(* Logix 5000 project; controller Bandas_Divert_Merge Emulate 5570 rev 30.12; software revision 30.00 *)

TASK MainTask (continuous, watchdog 500 ms) : MainProgram

MODULES
   Local : Emulate 5570 (ICP 2, rev 30.12)
      VIRTUAL_OUTPUTS : vendor 1 type 0 code 15 (ICP 4, rev 1.1, Output RPI 50 ms)   // Salidas_PLC_Bandas
      VIRTUAL_INPUTS : vendor 1 type 0 code 15 (ICP 3, rev 1.1, Output RPI 50 ms)   // Entradas_PLC_Bandas_Transportadoras
END_MODULES

VAR_GLOBAL   (* controller tags *)
   B1 : BOOL;
   B11 : BOOL;
   B2A : BOOL;
   B2A1 : BOOL;   // Banda hacia arriba
   B2B : BOOL;
   B2B1 : BOOL;   // Banda hacia izquierda
   B4A : BOOL;   // Banda4A
   B4B : BOOL;   // Banda4B
   B6A : BOOL;   // banda6A
   B6B : BOOL;   // banda 6b
   B_decA : BOOL;
   B_decB : BOOL;
   B_secA : BOOL;
   B_secB : BOOL;
   P : BOOL;   // Selector de baldosas
   Press_ActLX : INT;
   Press_ActLY : INT;
   Press_CilinderMax : BOOL;
   Press_CilinderMin : BOOL;
   Press_CilinderPos : INT;
   Press_FillerMax : BOOL;
   Press_FillerMin : BOOL;
   Press_FillerPos : INT;
   Press_Manguera : BOOL;
   Press_SourceTiles : BOOL;
   Press_SXmax : BOOL;
   Press_SXmin : BOOL;
   Press_TileMax : BOOL;
   Press_TileMin : BOOL;
   Press_TilePos : INT;
   Press_Ymax : BOOL;
   Press_Ymin : BOOL;
   S1 : BOOL;
   S11 : BOOL;
   S2 : BOOL;
   S21 : BOOL;
   S4 : BOOL;   // Sensor4_Para la engobadora
   S6 : BOOL;   // Sensor6_Va para el merge
   S_dec : BOOL;
   S_sec : BOOL;
   SFC_Bder4 : BOOL;
   SFC_Bizq4 : BOOL;
   SFC_BunionX : BOOL;
   SFC_BunionY : BOOL;
   SFC_Sder4 : BOOL;
   SFC_Sizq4 : BOOL;
   SFC_Sunion : BOOL;
   Start : BOOL;
   Tipper_Grab : INT;
   Tipper_Rollers : BOOL;
   Tipper_Rotate : INT;
   Tipper_S1 : BOOL;
   Tipper_S2 : BOOL;
END_VAR

PROGRAM MainProgram   (* main routine MainRoutine *)
VAR
   Action_000 : SFC_ACTION := (Status := 16#0020_0000, PauseTimer := 1);
   Action_001 : SFC_ACTION := (Status := 16#0020_0000, PauseTimer := 1);
   Action_002 : SFC_ACTION := (Status := 16#0020_0000, PauseTimer := 1);
   Action_003 : SFC_ACTION := (Status := 16#0020_0000, PauseTimer := 1);
   Action_004 : SFC_ACTION := (Status := 16#0020_0000, PauseTimer := 1);
   Action_005 : SFC_ACTION := (Status := 16#0020_0000, PauseTimer := 1);
   Action_006 : SFC_ACTION := (Status := 16#0020_0000, PauseTimer := 1);
   Action_007 : SFC_ACTION := (Status := 16#0020_0000, PauseTimer := 1);
   Action_008 : SFC_ACTION := (Status := 16#0020_0000, PauseTimer := 1);
   Action_009 : SFC_ACTION := (Status := 16#0020_0000, PauseTimer := 1);
   Action_010 : SFC_ACTION := (Status := 16#0020_0000, PauseTimer := 1);
   Action_011 : SFC_ACTION := (Status := 16#0020_0000, PauseTimer := 1);
   Action_012 : SFC_ACTION := (Status := 16#0020_0000, PauseTimer := 1);
   Action_013 : SFC_ACTION := (Status := 16#0020_0000, PauseTimer := 1);
   Action_014 : SFC_ACTION := (Status := 16#0020_0000, PauseTimer := 1);
   Action_015 : SFC_ACTION := (Status := 16#0020_0000, PauseTimer := 1);
   Action_016 : SFC_ACTION := (Status := 16#0020_0000, PauseTimer := 1);
   Action_017 : SFC_ACTION := (Status := 16#0020_0000, PauseTimer := 1);
   Action_018 : SFC_ACTION := (Status := 16#0020_0000, PauseTimer := 1);
   Action_019 : SFC_ACTION := (Status := 16#0020_0000, PauseTimer := 1);
   Action_020 : SFC_ACTION := (Status := 16#0020_0000, PauseTimer := 1);
   Action_021 : SFC_ACTION := (Status := 16#0020_0000, PauseTimer := 1);
   Action_022 : SFC_ACTION := (Status := 16#0020_0000, PauseTimer := 1);
   Action_023 : SFC_ACTION := (Status := 16#0020_0000, PauseTimer := 1);
   Action_024 : SFC_ACTION := (Status := 16#0020_0000, PauseTimer := 1);
   Action_025 : SFC_ACTION := (Status := 16#0020_0000, PauseTimer := 1);
   Action_026 : SFC_ACTION := (Status := 16#0020_0000, PauseTimer := 1);
   Action_027 : SFC_ACTION := (Status := 16#0020_0000, PauseTimer := 1);
   Action_028 : SFC_ACTION := (Status := 16#0020_0000, PauseTimer := 1);
   Action_029 : SFC_ACTION := (Status := 16#0020_0000, PauseTimer := 1);
   Action_030 : SFC_ACTION := (Status := 16#0020_0000, PauseTimer := 1);
   Action_031 : SFC_ACTION := (Status := 16#0020_0000, PauseTimer := 1);
   Action_032 : SFC_ACTION := (Status := 16#0020_0000, PauseTimer := 1);
   Action_033 : SFC_ACTION := (Status := 16#0020_0000, PauseTimer := 1);
   Action_034 : SFC_ACTION := (Status := 16#0020_0000, PauseTimer := 1);
   B1 : BOOL;
   B2A : BOOL;   // Banda hacia arriba
   B2B : BOOL;   // Banda hacia izquierda
   B4A : BOOL;   // Banda4A
   B4B : BOOL;   // Banda4B
   B6A : BOOL;   // banda6A
   B6B : BOOL;   // banda 6b
   B_decA : BOOL;
   B_decB : BOOL;
   B_secA : BOOL;
   B_secB : BOOL;
   Bandera1 : BOOL;
   Bandera2 : BOOL;
   Bandera3 : BOOL;
   Bandera4 : BOOL;
   Bandera5 : BOOL;
   Bandera7 : BOOL;
   Bandera7X : BOOL;
   Bandera7y : BOOL;
   Bandera8 : BOOL;
   Bandera9 : BOOL;
   C1 : COUNTER := (PRE := 4);   // Contador banda 1
   C2 : COUNTER := (PRE := 4);   // Contador banda 2
   Contador1 : COUNTER := (PRE := 2);
   FB_Sensor_Bandera7 : BOOL;
   FB_Sensor_Bifurcado : BOOL;
   FB_Sensor_Principal : BOOL;
   FB_SensorI1 : BOOL;
   P : BOOL;   // Selección en la bifurcacion
   ResetC1 : BOOL;
   ResetC2 : BOOL;
   S1 : BOOL;
   S2 : BOOL;
   S4 : BOOL;   // Sensor4_Para la engobadora
   S6 : BOOL;   // Sensor6_Va para el merge
   S_dec : BOOL;
   S_sec : BOOL;
   SelP : BOOL := 1;   // Seleccionar botón
   Sensor_Bandera7 : BOOL;
   Sensor_Bifurcado : BOOL;
   Sensor_Principal : BOOL;
   SensorI1 : BOOL;
   Start : BOOL;
   StartRoutine : BOOL := 1;
   Step_000 : SFC_STEP := (Status := 16#0020_0000, PauseTimer := 1);
   Step_001 : SFC_STEP := (Status := 16#0020_0000, PauseTimer := 1);
   Step_002 : SFC_STEP := (Status := 16#0020_0000, PauseTimer := 1);
   Step_003 : SFC_STEP := (Status := 16#0020_0000, PauseTimer := 1);
   Step_004 : SFC_STEP := (Status := 16#0020_0000, PauseTimer := 1);
   Step_005 : SFC_STEP := (Status := 16#0020_0000, PauseTimer := 1);
   Step_006 : SFC_STEP := (Status := 16#0020_0000, PauseTimer := 1);
   Step_007 : SFC_STEP := (Status := 16#0020_0000, PauseTimer := 1);
   Step_008 : SFC_STEP := (Status := 16#0020_0000, PauseTimer := 1);
   Step_009 : SFC_STEP := (Status := 16#0020_0000, PauseTimer := 1);
   Step_010 : SFC_STEP := (Status := 16#0020_0000, PauseTimer := 1);
   Step_011 : SFC_STEP := (Status := 16#0020_0000, PauseTimer := 1);
   Step_012 : SFC_STEP := (Status := 16#0020_0000, PauseTimer := 1);
   Step_013 : SFC_STEP := (Status := 16#0020_0000, PauseTimer := 1);
   Step_014 : SFC_STEP := (Status := 16#0020_0000, PauseTimer := 1);
   Step_015 : SFC_STEP := (Status := 16#0020_0000, PauseTimer := 1);
   Step_016 : SFC_STEP := (Status := 16#0020_0000, PauseTimer := 1);
   Step_017 : SFC_STEP := (Status := 16#0020_0000, PauseTimer := 1);
   Step_018 : SFC_STEP := (Status := 16#0020_0000, PauseTimer := 1);
   Step_019 : SFC_STEP := (Status := 16#0020_0000, PauseTimer := 1);
   Step_020 : SFC_STEP := (Status := 16#0020_0000, PauseTimer := 1);
   Step_021 : SFC_STEP := (Status := 16#0020_0000, PauseTimer := 1);
   Step_022 : SFC_STEP := (Status := 16#0020_0000, PauseTimer := 1);
   Step_023 : SFC_STEP := (Status := 16#0020_0000, PauseTimer := 1, PRE := 500);
   Step_024 : SFC_STEP := (Status := 16#0020_0000, PauseTimer := 1);
   Step_025 : SFC_STEP := (Status := 16#0020_0000, PauseTimer := 1);
   Step_026 : SFC_STEP := (Status := 16#0020_0000, PauseTimer := 1);
   Step_027 : SFC_STEP := (Status := 16#0020_0000, PauseTimer := 1, PRE := 200);
   Step_028 : SFC_STEP := (Status := 16#0020_0000, PauseTimer := 1);
   Step_029 : SFC_STEP := (Status := 16#0020_0000, PauseTimer := 1);
   Step_030 : SFC_STEP := (Status := 16#0020_0000, PauseTimer := 1);
   Step_031 : SFC_STEP := (Status := 16#0020_0000, PauseTimer := 1, PRE := 5000);
   Step_032 : SFC_STEP := (Status := 16#0020_0000, PauseTimer := 1);
   Step_033 : SFC_STEP := (Status := 16#0020_0000, PauseTimer := 1);
   Step_034 : SFC_STEP := (Status := 16#0020_0000, PauseTimer := 1);
   Step_035 : SFC_STEP := (Status := 16#0020_0000, PauseTimer := 1);
   Step_036 : SFC_STEP := (Status := 16#0020_0000, PauseTimer := 1);
   Step_037 : SFC_STEP := (Status := 16#0020_0000, PauseTimer := 1);
   Step_038 : SFC_STEP := (Status := 16#0020_0000, PauseTimer := 1);
   Step_039 : SFC_STEP := (Status := 16#0020_0000, PauseTimer := 1);
   Step_040 : SFC_STEP := (Status := 16#0020_0000, PauseTimer := 1);
   Step_041 : SFC_STEP := (Status := 16#0020_0000, PauseTimer := 1);
   Step_042 : SFC_STEP := (Status := 16#0020_0000, PauseTimer := 1);
   Step_043 : SFC_STEP := (Status := 16#0020_0000, PauseTimer := 1);
   Step_044 : SFC_STEP := (Status := 16#0020_0000, PauseTimer := 1);
   Step_045 : SFC_STEP := (Status := 16#0020_0000, PauseTimer := 1);
   Step_046 : SFC_STEP := (Status := 16#0020_0000, PauseTimer := 1, PRE := 200);
   Step_051 : SFC_STEP := (Status := 16#0020_0000, PauseTimer := 1, PRE := 200);
   Stop : BOOL;
   Tran_000 : BOOL;
   Tran_001 : BOOL;
   Tran_002 : BOOL;
   Tran_003 : BOOL;
   Tran_004 : BOOL;
   Tran_005 : BOOL;
   Tran_006 : BOOL;
   Tran_007 : BOOL;
   Tran_008 : BOOL;
   Tran_009 : BOOL;
   Tran_010 : BOOL;
   Tran_011 : BOOL;
   Tran_012 : BOOL;
   Tran_013 : BOOL;
   Tran_014 : BOOL;
   Tran_015 : BOOL;
   Tran_016 : BOOL;
   Tran_017 : BOOL;
   Tran_018 : BOOL;
   Tran_019 : BOOL;
   Tran_020 : BOOL;
   Tran_021 : BOOL;
   Tran_022 : BOOL;
   Tran_023 : BOOL;
   Tran_024 : BOOL;
   Tran_025 : BOOL;
   Tran_026 : BOOL;
   Tran_027 : BOOL;
   Tran_028 : BOOL;
   Tran_029 : BOOL;
   Tran_030 : BOOL;
   Tran_031 : BOOL;
   Tran_032 : BOOL;
   Tran_033 : BOOL;
   Tran_034 : BOOL;
   Tran_035 : BOOL;
   Tran_036 : BOOL;
   Tran_037 : BOOL;
   Tran_038 : BOOL;
   Tran_039 : BOOL;
   Tran_040 : BOOL;
   Tran_041 : BOOL;
   Tran_042 : BOOL;
   Tran_043 : BOOL;
   Tran_044 : BOOL;
   Tran_045 : BOOL;
   Tran_046 : BOOL;
   Tran_047 : BOOL;
   Tran_048 : BOOL;
   Tran_049 : BOOL;
END_VAR

ROUTINE MainRoutine   (* ladder *)
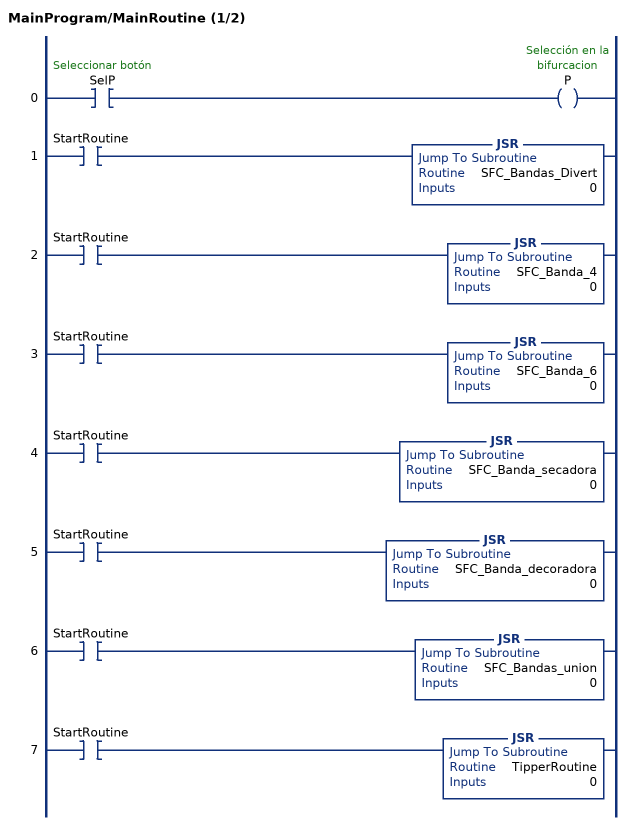
   0: XIC(SelP)OTE(P);
   1: XIC(StartRoutine)JSR(SFC_Bandas_Divert,0);
   2: XIC(StartRoutine)JSR(SFC_Banda_4,0);
   3: XIC(StartRoutine)JSR(SFC_Banda_6,0);
   4: XIC(StartRoutine)JSR(SFC_Banda_secadora,0);
   5: XIC(StartRoutine)JSR(SFC_Banda_decoradora,0);
   6: XIC(StartRoutine)JSR(SFC_Bandas_union,0);
   7: XIC(StartRoutine)JSR(TipperRoutine,0);
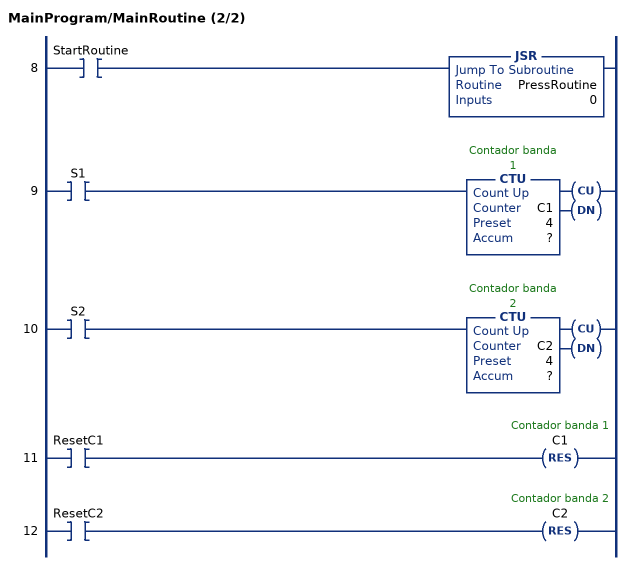
   8: XIC(StartRoutine)JSR(PressRoutine,0);
   9: XIC(S1)CTU(C1,?,?);
   10: XIC(S2)CTU(C2,?,?);
   11: XIC(ResetC1)RES(C1);
   12: XIC(ResetC2)RES(C2);
END_ROUTINE

ROUTINE PressRoutine   (* sequential function chart *)
// Rutina prensa
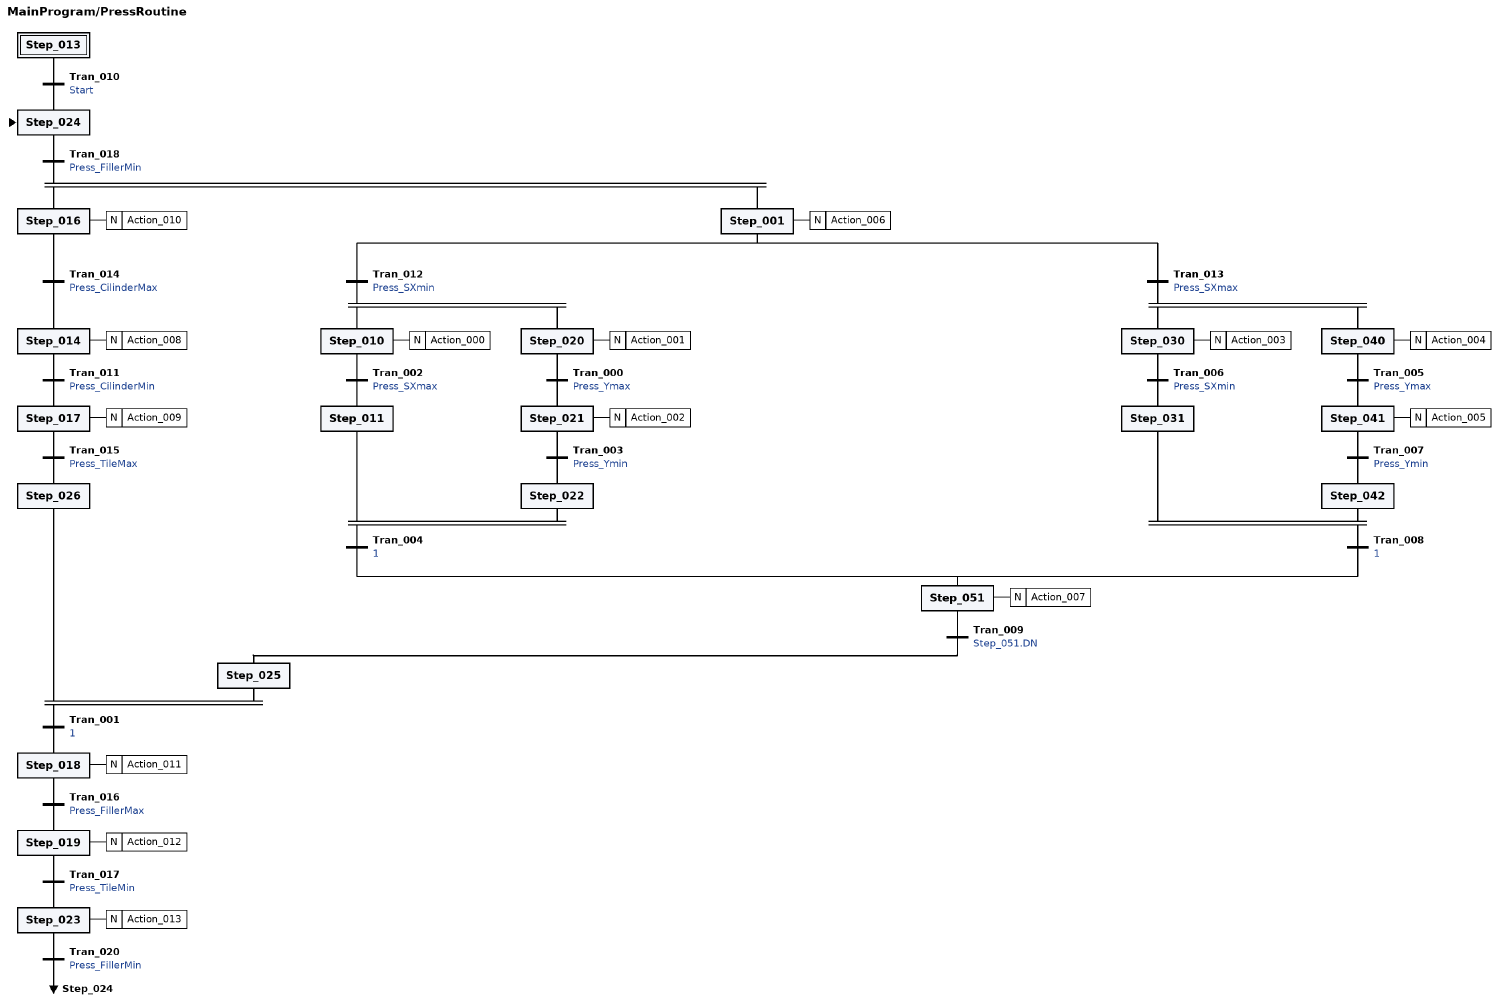
   INITIAL_STEP Step_013:
   END_STEP
   TRANSITION Tran_010 FROM Step_013 TO Step_024
      := Start
   END_TRANSITION
   STEP Step_024:
   END_STEP
   TRANSITION Tran_018 FROM Step_024 TO (Step_016, Step_001)
      := Press_FillerMin
   END_TRANSITION
   STEP Step_016:
      ACTION Action_010 (N):
         Press_CilinderPos := 140;
         Press_SourceTiles :=1;
      END_ACTION
   END_STEP
   STEP Step_001:
      ACTION Action_006 (N):
         Press_Manguera :=1;
      END_ACTION
   END_STEP
   TRANSITION Tran_014 FROM Step_016 TO Step_014
      := Press_CilinderMax
   END_TRANSITION
   TRANSITION Tran_012 FROM Step_001 TO (Step_020, Step_010)
      := Press_SXmin
   END_TRANSITION
   TRANSITION Tran_013 FROM Step_001 TO (Step_040, Step_030)
      := Press_SXmax
   END_TRANSITION
   STEP Step_014:
      ACTION Action_008 (N):
         Press_SourceTiles :=0;
         Press_CilinderPos := 0;
         
      END_ACTION
   END_STEP
   TRANSITION Tran_011 FROM Step_014 TO Step_017
      := Press_CilinderMin
         
   END_TRANSITION
   STEP Step_010:
      ACTION Action_000 (N):
         Press_ActLX := 1220;
      END_ACTION
   END_STEP
   STEP Step_020:
      ACTION Action_001 (N):
         Press_ActLY := 710;
      END_ACTION
   END_STEP
   STEP Step_017:
      ACTION Action_009 (N):
         Press_TilePos := 9;
      END_ACTION
   END_STEP
   STEP Step_030:
      ACTION Action_003 (N):
         Press_ActLX := 0;
      END_ACTION
   END_STEP
   STEP Step_040:
      ACTION Action_004 (N):
         Press_ActLY := 710;
      END_ACTION
   END_STEP
   TRANSITION Tran_002 FROM Step_010 TO Step_011
      := Press_SXmax
   END_TRANSITION
   TRANSITION Tran_000 FROM Step_020 TO Step_021
      := Press_Ymax
   END_TRANSITION
   TRANSITION Tran_015 FROM Step_017 TO Step_026
      := Press_TileMax
         
   END_TRANSITION
   TRANSITION Tran_006 FROM Step_030 TO Step_031
      := Press_SXmin
   END_TRANSITION
   TRANSITION Tran_005 FROM Step_040 TO Step_041
      := Press_Ymax
   END_TRANSITION
   STEP Step_021:
      ACTION Action_002 (N):
         Press_ActLY := 0;
         
      END_ACTION
   END_STEP
   STEP Step_026:
   END_STEP
   STEP Step_025:
   END_STEP
   STEP Step_041:
      ACTION Action_005 (N):
         Press_ActLY := 0;
      END_ACTION
   END_STEP
   TRANSITION Tran_003 FROM Step_021 TO Step_022
      := Press_Ymin
   END_TRANSITION
   TRANSITION Tran_007 FROM Step_041 TO Step_042
      := Press_Ymin
   END_TRANSITION
   TRANSITION Tran_001 FROM (Step_025, Step_026) TO Step_018
      := 1
   END_TRANSITION
   STEP Step_011:
   END_STEP
   STEP Step_022:
   END_STEP
   STEP Step_031:
   END_STEP
   STEP Step_042:
   END_STEP
   STEP Step_018:
      ACTION Action_011 (N):
         Press_FillerPos := 800;
      END_ACTION
   END_STEP
   TRANSITION Tran_004 FROM (Step_011, Step_022) TO Step_051
      := 1
   END_TRANSITION
   TRANSITION Tran_008 FROM (Step_031, Step_042) TO Step_051
      := 1
   END_TRANSITION
   TRANSITION Tran_016 FROM Step_018 TO Step_019
      := Press_FillerMax
   END_TRANSITION
   STEP Step_019:
      ACTION Action_012 (N):
         Press_TilePos := 0;
      END_ACTION
   END_STEP
   STEP Step_051:
      ACTION Action_007 (N):
         Press_Manguera :=0;
      END_ACTION
   END_STEP
   TRANSITION Tran_017 FROM Step_019 TO Step_023
      := Press_TileMin
         
   END_TRANSITION
   TRANSITION Tran_009 FROM Step_051 TO Step_025
      := Step_051.DN
   END_TRANSITION
   STEP Step_023:
      ACTION Action_013 (N):
         Press_FillerPos := 0;
      END_ACTION
   END_STEP
   TRANSITION Tran_020 FROM Step_023 TO Step_024
      := Press_FillerMin
         
   END_TRANSITION
END_ROUTINE

ROUTINE SFC_Banda_4   (* sequential function chart *)
// Para rotar las baldosas por el camino del engobe
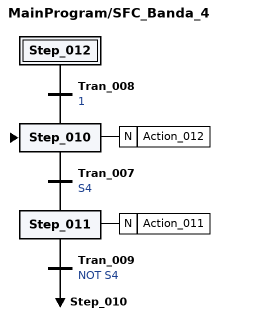
   INITIAL_STEP Step_012:
   END_STEP
   TRANSITION Tran_008 FROM Step_012 TO Step_010
      := 1
   END_TRANSITION
   STEP Step_010:
      ACTION Action_012 (N):
         B4A:=0;
         B4B:=1;
         
      END_ACTION
   END_STEP
   TRANSITION Tran_007 FROM Step_010 TO Step_011
      := S4
         
   END_TRANSITION
   STEP Step_011:
      ACTION Action_011 (N):
         B4A:=1;
         B4B:=0;
         
      END_ACTION
   END_STEP
   TRANSITION Tran_009 FROM Step_011 TO Step_010
      := NOT S4
   END_TRANSITION
END_ROUTINE

ROUTINE SFC_Banda_6   (* sequential function chart *)
// banda 6 que va después de la esmaltadora
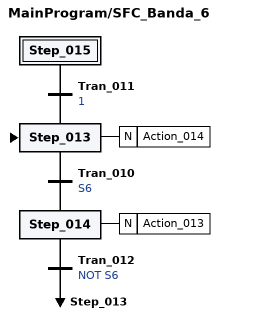
   INITIAL_STEP Step_015:
   END_STEP
   TRANSITION Tran_011 FROM Step_015 TO Step_013
      := 1
   END_TRANSITION
   STEP Step_013:
      ACTION Action_014 (N):
         B6A:=0;
         B6B:=1;
         
      END_ACTION
   END_STEP
   TRANSITION Tran_010 FROM Step_013 TO Step_014
      := S6
   END_TRANSITION
   STEP Step_014:
      ACTION Action_013 (N):
         B6A:=1;
         B6B:=0;
         
      END_ACTION
   END_STEP
   TRANSITION Tran_012 FROM Step_014 TO Step_013
      := NOT S6
   END_TRANSITION
END_ROUTINE

ROUTINE SFC_Banda_decoradora   (* sequential function chart *)
// Girar baldosas después de la decoradora hacia el horno
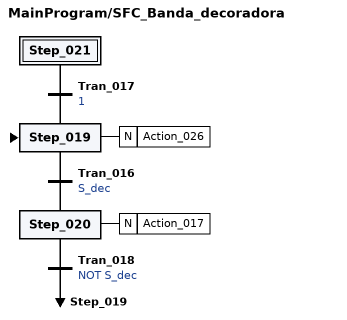
   INITIAL_STEP Step_021:
   END_STEP
   TRANSITION Tran_017 FROM Step_021 TO Step_019
      := 1
   END_TRANSITION
   STEP Step_019:
      ACTION Action_026 (N):
         B_decA:=0;
         B_decB:=1;
         
      END_ACTION
   END_STEP
   TRANSITION Tran_016 FROM Step_019 TO Step_020
      := S_dec
         
   END_TRANSITION
   STEP Step_020:
      ACTION Action_017 (N):
         B_decA:=1;
         B_decB:=0;
         
      END_ACTION
   END_STEP
   TRANSITION Tran_018 FROM Step_020 TO Step_019
      := NOT S_dec
         
   END_TRANSITION
END_ROUTINE

ROUTINE SFC_Banda_secadora   (* sequential function chart *)
// Para rotar las baldosas después de la secadora
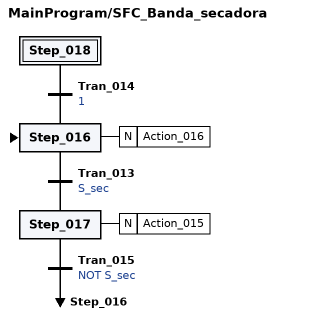
   INITIAL_STEP Step_018:
   END_STEP
   TRANSITION Tran_014 FROM Step_018 TO Step_016
      := 1
   END_TRANSITION
   STEP Step_016:
      ACTION Action_016 (N):
         B_secA:=0;
         B_secB:=1;
         
      END_ACTION
   END_STEP
   TRANSITION Tran_013 FROM Step_016 TO Step_017
      := S_sec
         
   END_TRANSITION
   STEP Step_017:
      ACTION Action_015 (N):
         B_secA:=1;
         B_secB:=0;
         
      END_ACTION
   END_STEP
   TRANSITION Tran_015 FROM Step_017 TO Step_016
      := NOT S_sec
         
   END_TRANSITION
END_ROUTINE

ROUTINE SFC_Bandas_Divert   (* sequential function chart *)
// Logica para mover las bandas entre maquinas
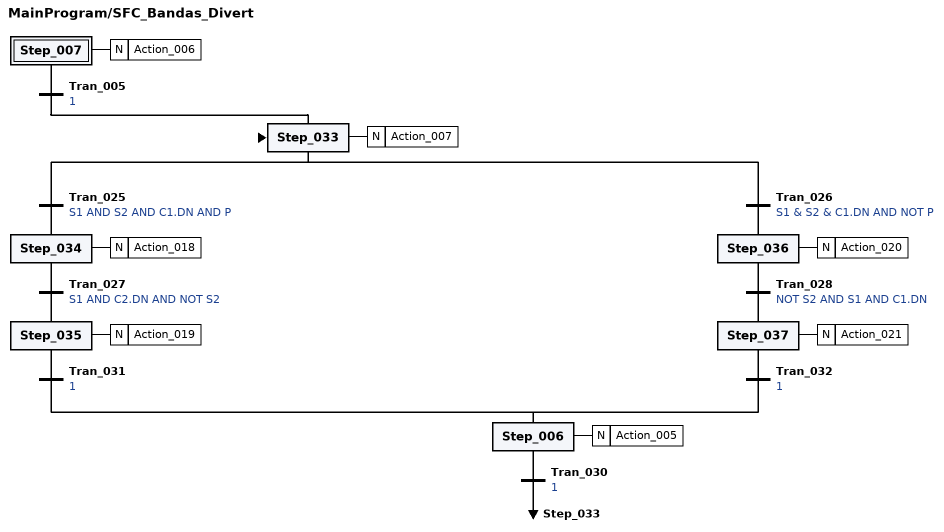
   INITIAL_STEP Step_007:
      ACTION Action_006 (N):
         B1 := 1;
         B2A := 1;
         B2B := 0;
      END_ACTION
   END_STEP
   TRANSITION Tran_005 FROM Step_007 TO Step_033
      := 1
   END_TRANSITION
   STEP Step_033:
      ACTION Action_007 (N):
         B1 := 1;
         B2A := 1;
         B2B := 0;
      END_ACTION
   END_STEP
   TRANSITION Tran_025 FROM Step_033 TO Step_034
      := S1 AND S2 AND C1.DN AND P
   END_TRANSITION
   TRANSITION Tran_026 FROM Step_033 TO Step_036
      := S1 & S2 & C1.DN AND NOT P
   END_TRANSITION
   STEP Step_034:
      ACTION Action_018 (N):
         B1 :=0;
         B2A :=1;
         B2B :=0;
      END_ACTION
   END_STEP
   STEP Step_036:
      ACTION Action_020 (N):
         B1 :=0;
         B2A :=0;
         B2B :=1;
      END_ACTION
   END_STEP
   TRANSITION Tran_027 FROM Step_034 TO Step_035
      := S1 AND C2.DN AND NOT S2
   END_TRANSITION
   TRANSITION Tran_028 FROM Step_036 TO Step_037
      := NOT S2 AND S1 AND C1.DN
   END_TRANSITION
   STEP Step_035:
      ACTION Action_019 (N):
         ResetC1 :=1;
         B1 := 1;
         B2A := 1;
         ResetC2 := 1;
      END_ACTION
   END_STEP
   STEP Step_037:
      ACTION Action_021 (N):
         ResetC1 := 1;
         B1 := 1;
         B2A := 1;
         ResetC2 := 1;
      END_ACTION
   END_STEP
   TRANSITION Tran_031 FROM Step_035 TO Step_006
      := 1
   END_TRANSITION
   TRANSITION Tran_032 FROM Step_037 TO Step_006
      := 1
   END_TRANSITION
   STEP Step_006:
      ACTION Action_005 (N):
         ResetC2 := 0;
         ResetC1 := 0;
      END_ACTION
   END_STEP
   TRANSITION Tran_030 FROM Step_006 TO Step_033
      := 1
   END_TRANSITION
END_ROUTINE

ROUTINE SFC_Bandas_union   (* sequential function chart *)
// Union merge bandas después de la decoradora
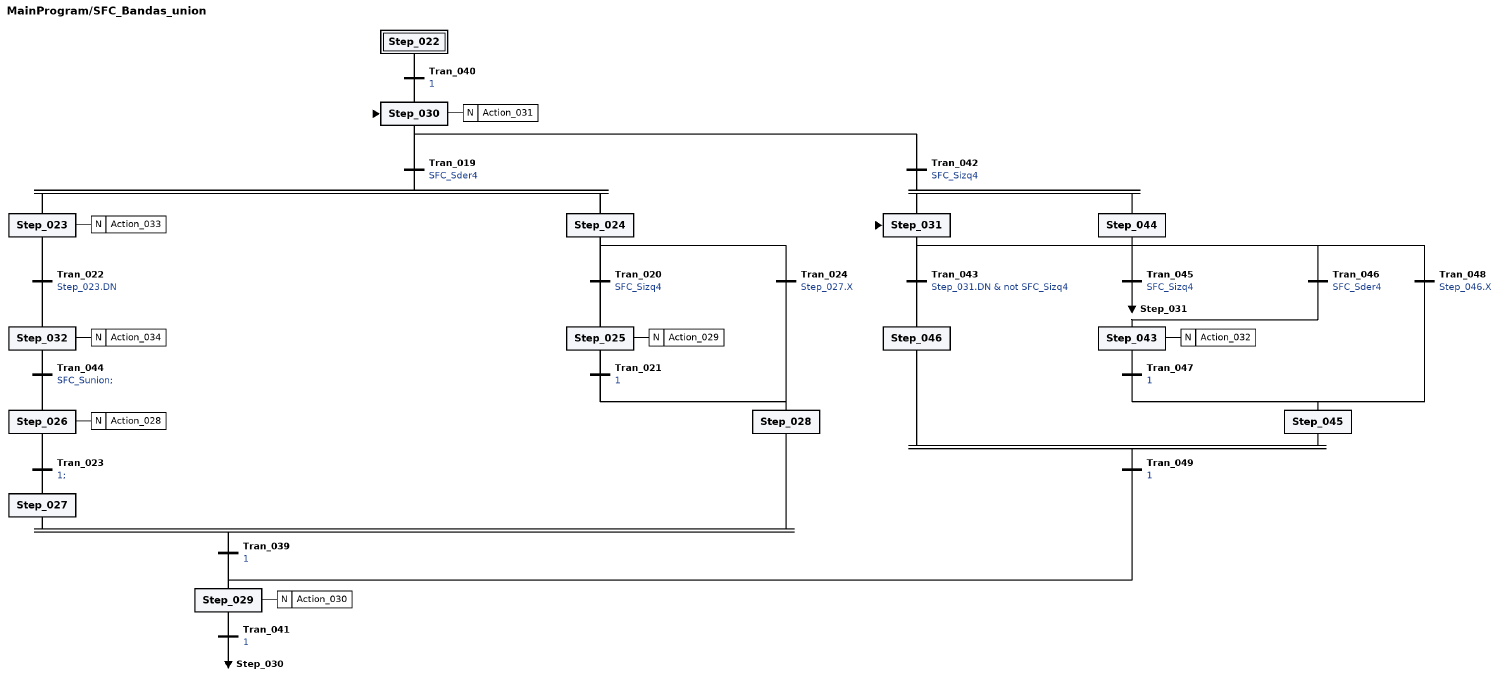
   INITIAL_STEP Step_022:
   END_STEP
   TRANSITION Tran_040 FROM Step_022 TO Step_030
      := 1
   END_TRANSITION
   STEP Step_030:
      ACTION Action_031 (N):
         SFC_Bder4:=1;
         SFC_Bizq4:=1;
         SFC_BunionX:=1;
      END_ACTION
   END_STEP
   TRANSITION Tran_019 FROM Step_030 TO (Step_024, Step_023)
      := SFC_Sder4
   END_TRANSITION
   TRANSITION Tran_042 FROM Step_030 TO (Step_044, Step_031)
      := SFC_Sizq4
   END_TRANSITION
   STEP Step_023:
      ACTION Action_033 (N):
         SFC_BunionY:=1;
         SFC_BunionX:=0;
      END_ACTION
   END_STEP
   STEP Step_024:
   END_STEP
   STEP Step_044:
   END_STEP
   TRANSITION Tran_022 FROM Step_023 TO Step_032
      := Step_023.DN
   END_TRANSITION
   STEP Step_032:
      ACTION Action_034 (N):
         SFC_Bder4:=0;
      END_ACTION
   END_STEP
   TRANSITION Tran_046 FROM Step_044 TO Step_043
      := SFC_Sder4
   END_TRANSITION
   STEP Step_031:
   END_STEP
   TRANSITION Tran_020 FROM Step_024 TO Step_025
      := SFC_Sizq4
   END_TRANSITION
   TRANSITION Tran_044 FROM Step_032 TO Step_026
      := SFC_Sunion;
   END_TRANSITION
   STEP Step_043:
      ACTION Action_032 (N):
         SFC_Bder4:=0;
      END_ACTION
   END_STEP
   STEP Step_025:
      ACTION Action_029 (N):
         SFC_Bizq4:=0;
      END_ACTION
   END_STEP
   TRANSITION Tran_048 FROM Step_044 TO Step_045
      := Step_046.X
   END_TRANSITION
   TRANSITION Tran_024 FROM Step_024 TO Step_028
      := Step_027.X
   END_TRANSITION
   STEP Step_026:
      ACTION Action_028 (N):
         SFC_BunionY:=0;
         
      END_ACTION
   END_STEP
   TRANSITION Tran_047 FROM Step_043 TO Step_045
      := 1
         
   END_TRANSITION
   TRANSITION Tran_045 FROM Step_031 TO Step_031
      := SFC_Sizq4
   END_TRANSITION
   TRANSITION Tran_021 FROM Step_025 TO Step_028
      := 1
         
   END_TRANSITION
   TRANSITION Tran_023 FROM Step_026 TO Step_027
      := 1;
   END_TRANSITION
   TRANSITION Tran_043 FROM Step_031 TO Step_046
      := Step_031.DN & not SFC_Sizq4
   END_TRANSITION
   STEP Step_045:
   END_STEP
   STEP Step_027:
   END_STEP
   STEP Step_028:
   END_STEP
   STEP Step_046:
   END_STEP
   TRANSITION Tran_039 FROM (Step_027, Step_028) TO Step_029
      := 1
         
   END_TRANSITION
   TRANSITION Tran_049 FROM (Step_045, Step_046) TO Step_029
      := 1
   END_TRANSITION
   STEP Step_029:
      ACTION Action_030 (N):
         SFC_BunionX:=1;
         SFC_Bizq4:=0;
      END_ACTION
   END_STEP
   TRANSITION Tran_041 FROM Step_029 TO Step_030
      := 1
         
   END_TRANSITION
END_ROUTINE

ROUTINE TipperRoutine   (* sequential function chart *)
// volteadora
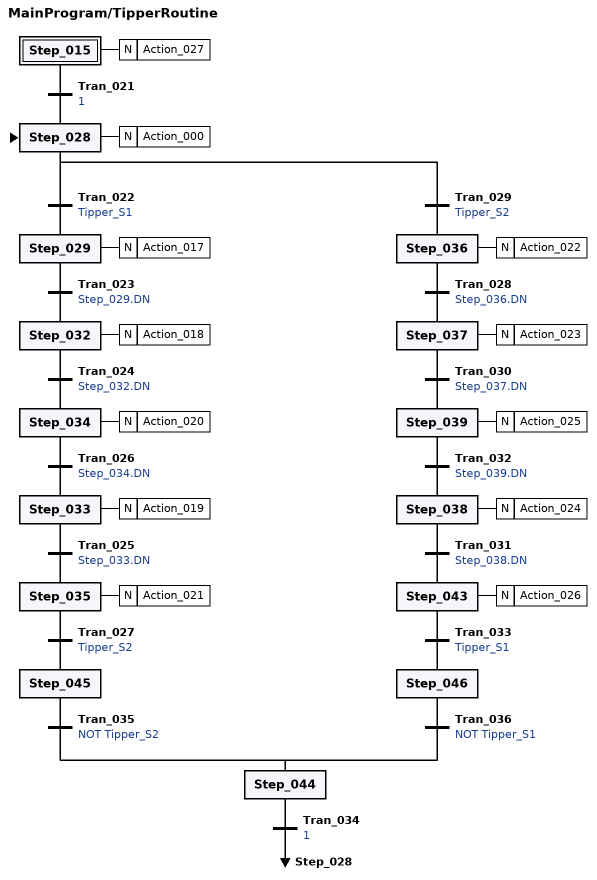
   INITIAL_STEP Step_015:
      ACTION Action_027 (N):
         Tipper_Rotate :=0;
      END_ACTION
   END_STEP
   TRANSITION Tran_021 FROM Step_015 TO Step_028
      := 1
         
   END_TRANSITION
   STEP Step_028:
      ACTION Action_000 (N):
         Tipper_Rollers :=1;
      END_ACTION
   END_STEP
   TRANSITION Tran_022 FROM Step_028 TO Step_029
      := Tipper_S1
   END_TRANSITION
   TRANSITION Tran_029 FROM Step_028 TO Step_036
      := Tipper_S2
         
   END_TRANSITION
   STEP Step_029:
      ACTION Action_017 (N):
         Tipper_Rollers :=0;
      END_ACTION
   END_STEP
   STEP Step_036:
      ACTION Action_022 (N):
         Tipper_Rollers :=0;
      END_ACTION
   END_STEP
   TRANSITION Tran_023 FROM Step_029 TO Step_032
      := Step_029.DN
   END_TRANSITION
   TRANSITION Tran_028 FROM Step_036 TO Step_037
      := Step_036.DN
   END_TRANSITION
   STEP Step_032:
      ACTION Action_018 (N):
         Tipper_Grab:=8;
      END_ACTION
   END_STEP
   STEP Step_037:
      ACTION Action_023 (N):
         Tipper_Grab:=8;
      END_ACTION
   END_STEP
   TRANSITION Tran_024 FROM Step_032 TO Step_034
      := Step_032.DN
   END_TRANSITION
   TRANSITION Tran_030 FROM Step_037 TO Step_039
      := Step_037.DN
   END_TRANSITION
   STEP Step_034:
      ACTION Action_020 (N):
         Tipper_Rotate:=180;
      END_ACTION
   END_STEP
   STEP Step_039:
      ACTION Action_025 (N):
         Tipper_Rotate:=0;
      END_ACTION
   END_STEP
   TRANSITION Tran_026 FROM Step_034 TO Step_033
      := Step_034.DN
   END_TRANSITION
   TRANSITION Tran_032 FROM Step_039 TO Step_038
      := Step_039.DN
   END_TRANSITION
   STEP Step_033:
      ACTION Action_019 (N):
         Tipper_Grab :=0;
      END_ACTION
   END_STEP
   STEP Step_038:
      ACTION Action_024 (N):
         Tipper_Grab :=0;
      END_ACTION
   END_STEP
   TRANSITION Tran_025 FROM Step_033 TO Step_035
      := Step_033.DN
   END_TRANSITION
   TRANSITION Tran_031 FROM Step_038 TO Step_043
      := Step_038.DN
   END_TRANSITION
   STEP Step_035:
      ACTION Action_021 (N):
         Tipper_Rollers :=1;
      END_ACTION
   END_STEP
   STEP Step_043:
      ACTION Action_026 (N):
         Tipper_Rollers :=1;
      END_ACTION
   END_STEP
   TRANSITION Tran_027 FROM Step_035 TO Step_045
      := Tipper_S2
   END_TRANSITION
   TRANSITION Tran_033 FROM Step_043 TO Step_046
      := Tipper_S1
   END_TRANSITION
   STEP Step_045:
   END_STEP
   STEP Step_046:
   END_STEP
   TRANSITION Tran_035 FROM Step_045 TO Step_044
      := NOT Tipper_S2
   END_TRANSITION
   TRANSITION Tran_036 FROM Step_046 TO Step_044
      := NOT Tipper_S1
   END_TRANSITION
   STEP Step_044:
   END_STEP
   TRANSITION Tran_034 FROM Step_044 TO Step_028
      := 1
   END_TRANSITION
END_ROUTINE
END_PROGRAM
